Universal Robots PolyScope program: PickPlaceAPS.urp

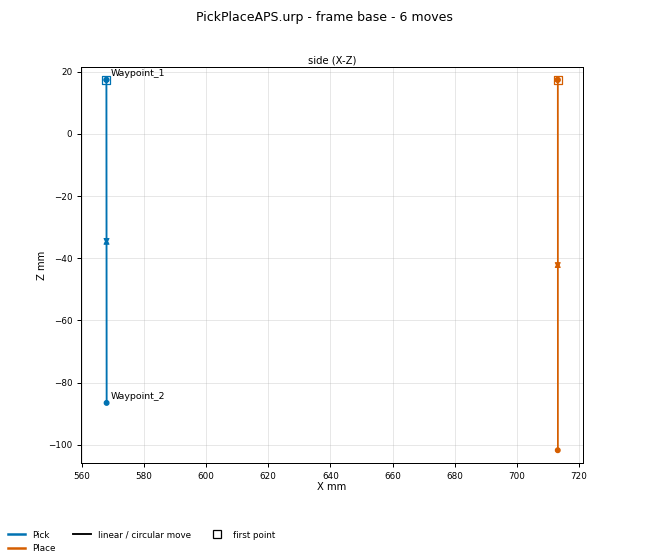
[picture p0: tool path of PickPlaceAPS.urp in frame base, 6 of 6 moves have a stored position in this frame; points joined in program order, loops and branches not executed]
Program PickPlaceAPS (installation=default directory=/programs/APS2OsUltimosRomanticos createdIn=3.15.3.106223 lastSavedIn=3.15.3.106223 robotSerialNumber=2017357017)
Calibrated DH parameters: a=[0.0001, -0.032836, -0.39033, 0.000086, 0.000053, 0]; d=[0.089393, 264.548863, -261.578988, -2.85966, 0.094927, 0.082356]; alpha=[1.569373, -0.001603, 0.013671, 1.570599, -1.570158, 0]; deltaTheta=[0.000031, -1.49356, 1.597104, -0.103695, -0.000023, -0.000043]
Robot Program (runOnlyOnce=false)
  Call Pick
  Call Place
SubProgram -> Pick
SubProgram -> Place
SubProgram Pick (keepSynchronizedWithDisk=false)
  MoveL speed 250 mm/s, acceleration 1200 mm/s^2 (useActiveTCP=true) feature=Base
    Waypoint Waypoint_1: TCP in base x=567.917 y=123.022 z=17.406 mm, rx=0.0447 ry=0.0138 rz=-0.0646 rad; joints [-180.013, -70.133, 102.031, -121.082, -86.78, 94.194] deg; flange x=570.416 y=114.885 z=197.204 mm, rx=-0.1009 ry=-3.1238 rz=-0.0699 rad
    Waypoint Waypoint_2: TCP in base x=567.969 y=122.941 z=-86.541 mm, rx=0.0446 ry=0.0137 rz=-0.0647 rad; joints [-180.053, -60.953, 107.189, -135.43, -86.929, 94.313] deg; flange x=570.453 y=114.821 z=93.259 mm, rx=-0.1011 ry=-3.1239 rz=-0.0698 rad
  Set DigitalOutput pin=tool_out[1]; digitalValue=0
  Set DigitalOutput pin=tool_out[0]; digitalValue=1
  Wait Sleep waitTime=0.5
  MoveL speed 250 mm/s, acceleration 1200 mm/s^2 (useActiveTCP=true) feature=Base
    Waypoint Waypoint_1: TCP in base x=567.917 y=123.022 z=17.406 mm, rx=0.0447 ry=0.0138 rz=-0.0646 rad; joints [-180.013, -70.133, 102.031, -121.082, -86.78, 94.194] deg; flange x=570.416 y=114.885 z=197.204 mm, rx=-0.1009 ry=-3.1238 rz=-0.0699 rad
SubProgram Place (keepSynchronizedWithDisk=false)
  MoveL speed 250 mm/s, acceleration 1200 mm/s^2 (useActiveTCP=true) feature=Base
    Waypoint Waypoint_3: TCP in base x=713.123 y=123.01 z=17.398 mm, rx=0.0447 ry=0.0138 rz=-0.0646 rad; joints [-180.023, -52.629, 74.353, -110.902, -86.721, 94.089] deg; flange x=715.624 y=114.872 z=197.197 mm, rx=-0.1009 ry=-3.1238 rz=-0.07 rad
    Waypoint Waypoint_4: TCP in base x=713.134 y=122.983 z=-101.774 mm, rx=0.0446 ry=0.0137 rz=-0.0646 rad; joints [-180.054, -44.735, 79.895, -124.346, -86.837, 94.219] deg; flange x=715.633 y=114.859 z=78.025 mm, rx=-0.1009 ry=-3.1238 rz=-0.0698 rad
  Set DigitalOutput pin=tool_out[1]; digitalValue=1
  Set DigitalOutput pin=tool_out[0]; digitalValue=0
  Wait Sleep waitTime=0.5
  MoveL speed 250 mm/s, acceleration 1200 mm/s^2 (useActiveTCP=true) feature=Base
    Waypoint Waypoint_3: TCP in base x=713.123 y=123.01 z=17.398 mm, rx=0.0447 ry=0.0138 rz=-0.0646 rad; joints [-180.023, -52.629, 74.353, -110.902, -86.721, 94.089] deg; flange x=715.624 y=114.872 z=197.197 mm, rx=-0.1009 ry=-3.1238 rz=-0.07 rad
